{attribute 'qualified_only'}
{attribute 'strict'}
{attribute 'to_string'}
TYPE E_RecipeRun :
(
	Initial := 1,		// 초기화 상태 (변수 초기화)
	Ramp := 2,			// Ramp 처리 상태 (현재 스텝의 동작 수행)
	CheckHoldTemp := 3,	// Hold Type 확인
	End := 5
);
END_TYPE

(* stored: Version 1.1.0.1, ProductVersion 3.1.4026.11
   DUT E_RecipeRun: Id {5e38f956-9195-425f-b108-a9af18eb5129} *)
